Staubli VAL3: create_easyCube.pgx

public program create_easyCube(point x_pOrigin, num x_nDistanceX, num x_nDistanceY, num x_nDistanceZ)
  local trsf l_trsfCopy
begin
  //
  // build the cube
  // Origin
  if setFrame(x_pOrigin,compose(x_pOrigin,world,{x_nDistanceX,0,0,0,0,0}),compose(x_pOrigin,world,{0,x_nDistanceY,0,0,0,0}),fCube)==0
    bCreate_cube=true
  else
    bCreate_cube=false
  endIf
  // Distance x y z
  nDistanceX_cube=x_nDistanceX
  nDistanceY_cube=x_nDistanceY
  nDistanceZ_cube=x_nDistanceZ
  // regolate the frame
  l_trsfCopy=fCube.trsf
  fCube.trsf={l_trsfCopy.x,l_trsfCopy.y,l_trsfCopy.z,0,0,0}
end
